FUNCTION_BLOCK bloco1
  (* Standard: 61499-2 *)
  (* Version 11-01-12, GASR *)
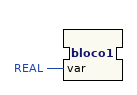
  VAR_INPUT
    var : REAL;
  END_VAR
  EC_STATES
    START;
  END_STATES
  ALGORITHM Alg1 IN Lua:
print('oi')
  END_ALGORITHM
END_FUNCTION_BLOCK
